PROGRAM DAQPassTime
VAR
	trigger					:BOOL	:= FALSE;
	tStart					:TIME; (* Time program start *)
    tWork 					:TIME; (* Execution time *)
END_VAR

IF GVL_DAQ.DAQ_CTR_INT.Measure_Run_Time AND NOT trigger THEN
	tStart											:= TIME();
	trigger											:= TRUE;
END_IF

IF NOT GVL_DAQ.DAQ_CTR_INT.Measure_Run_Time AND trigger THEN
	GVL_DAQ.RUNTIME_COLLECTOR[GVL_DAQ.PASS_INDEX]	:= TIME() - tStart;
	trigger											:= FALSE;
END_IF

END_PROGRAM

(* stored: Version 1.1.0.1, ProductVersion 3.1.4026.12
   POU DAQPassTime: Id {a9070ee4-2ede-45c9-ba05-e876686590a5}, SpecialFunc None *)
